PROGRAM MAIN
VAR
	PumpControl01				:	PumpControl01;
	PumpControl02				:	PumpControl02;
	M1_01: BOOL;
	M2_01: BOOL;
	M1_02: BOOL;
	M2_02: BOOL;
END_VAR

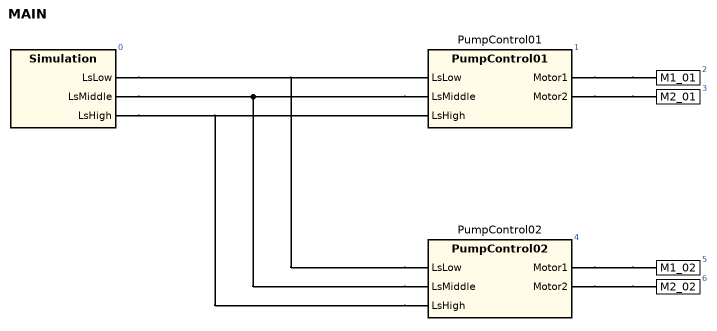
Simulation();
PumpControl01(LsLow := Simulation.LsLow, LsMiddle := Simulation.LsMiddle, LsHigh := Simulation.LsHigh);
M1_01 := PumpControl01.Motor1;
M2_01 := PumpControl01.Motor2;
PumpControl02(LsLow := Simulation.LsLow, LsMiddle := Simulation.LsMiddle, LsHigh := Simulation.LsHigh);
M1_02 := PumpControl02.Motor1;
M2_02 := PumpControl02.Motor2;

END_PROGRAM

(* stored: Version 1.1.0.1, ProductVersion 3.1.4024.15
   POU MAIN: Id {d5fd86cf-f8e9-4366-b8f5-17a052dcfb8a}, SpecialFunc None *)
